// TwinCAT 3 PLC project Untitled1
// ProgramVersion: 3.1.4024.0
// libraries:
//   Tc2_MC2, * (Beckhoff Automation GmbH)
//   Tc2_Standard, * (Beckhoff Automation GmbH)
//   Tc2_System, * (Beckhoff Automation GmbH)
//   Tc3_Module, * (Beckhoff Automation GmbH)
// project tree:
//   DUTs/ ST_AchsAuftrg.TcDUT, ST_AchsFreigb.TcDUT (not stored), ST_AchsGrdfkt.TcDUT (not stored), ST_AchsInOut.TcDUT, ST_AchsKoppln.TcDUT (not stored), ST_AchsParam.TcDUT, ST_AchsStatus.TcDUT, ST_MeldServoSchrauber_1.TcDUT, ST_NcAchsen.TcDUT, ST_ParamSKSServoschrauber.TcDUT
//   GVLs/ GlobalVar_NcAchsen.TcGVL
//   / PlcTask.TcTTO (not stored)
//   POUs/10_Funktionen/Diverse/ FB_LogFile_Schrauber.TcPOU (not stored), FB_Mittelwert.TcPOU (not stored)
//   POUs/10_Funktionen/History/ FB_StepHistory.TcPOU
//   POUs/10_Funktionen/SchraubBearb/Obj/ FB_Obj_Error_Schrauber.TcPOU (not stored), FB_Obj_IOSchlauch.TcPOU (not stored)
//   POUs/ FB_Schrauber_PnP.TcPOU (not stored), FB_Schrauber_PnP_Neu.TcPOU (not stored)

// ---- DUTs/ST_AchsAuftrg.TcDUT
TYPE ST_AchsAuftrg :
STRUCT
	// Achs-Fahrauftrag
	sPTP_AuftrgTyp		:STRING(15);	// Beschreibung des Achstyp. Standard, Endlos oder Modulo
	
	bPTP_PosiFrg		:BOOL;	// Achse hat die Freigabe zu Positionieren. Betriebsbereit, beide Vorschubfreigaben und kein anderer Achsstart steht an.

	fPTP_ZielPos		:LREAL;	// aktuelle Zielposition für den Achsfahrauftrag
	fPTP_LetzZiel		:LREAL;	// Zu letzt angefahrene Zielposition
	fPTP_Geschw			:LREAL;	// in %
	ePTP_BuffMode		:MC_BufferMode;	(*MC_Aborting,
												  MC_Buffered,
												  MC_BlendingLow,
												  MC_BlendingPrevious,
												  MC_BlendingNext,
												  MC_BlendingHigh*)
	arrPTP_start		:ARRAY[1..3] OF BOOL;	// Achsstart für 3 verschiedene Betriebsmodi. Definiert in E_AchsFahrauftraege oder in NcParameter als Konstante
	bPTP_aktiv			:BOOL;	// Achsauftrag ist gestartet und auch aktiv
	bPTP_inZiel			:BOOL;	// Achsauftrag ist gestartet und im Ziel. Gibt es bei Endlosbetrieb nicht. Wird bei Verwendung vom FB_AchsStartAusf sofort wieder FALSE
	bPTP_inFenst		:BOOL;	// Achsauftrag ist gestartet und im Ziel +- 0.1 Grad oder mm. Gibt es bei Endlosbetrieb nicht.
	bPTP_stop			:BOOL;	// Achsauftrag wird gestoppt. Wird bei Verwendung vom FB_AchsStartAusf ggf. überschrieben
	bPTP_Autostop		:BOOL;	// wird aktuell nicht verwendet
	bPTP_gest			:BOOL;	// Achsauftrag wurde gestoppt. Ist nur bei aktivem bPTP_stop TRUE. Bedeutet, dass auch hier der FB_AchsStartAusf das überschreiben könnte
	bPTP_halt			:BOOL;	// Override auf 0%. Es wird mit der Beschleunigung aus dem Systemmanager gerampt
	bPTP_verz			:BOOL;	// Override auf den Wert aus der Freig-Struktur setzen.
END_STRUCT
END_TYPE

// ---- DUTs/ST_AchsInOut.TcDUT
TYPE ST_AchsInOut :
STRUCT
	
	// Eingänge
	// #######################################################################
	I_nEinspeiseStatusword			AT %I*: WORD;	(*S-0-01720.0.2
										Bit 0 - 3 	-> reserviert
										Bit 4			-> Netzspannung OK
										Bit 5			-> Hardware bereit zum Einschalten
										Bit 6			-> Zwischenkreis wird gerade geladen, oder ist geladen
										Bit 8-9		-> Rückmeldung Betriebsart
										Bit 10		-> Zwischenkreisentladung angewählt und Zwischenkreis spannungsfrei (< ca. 35 V)
										Bit 11		-> Bremswiderstand aktiv
										Bit 12		-> Warnung aktiv
										Bit 13		-> Fehler aktiv
										Bit 14		-> Bereit zur Freigabe: Netzschütz geschlossen, Zwischenkreis geladen. Die versorgten Achsen zeigen "bb".
										Bit 15		-> Die Freigabe ist gegeben, d.h. der Zwischenkreis ist belastbar. Die versorgten Achsen können nach "Ab" geschaltet werden und die Antriebsfreigabe kann gesetzt werden.
															Bei den Wechselrichtern XM* muss das Bit von der Steuerung beschrieben werden, wenn der Versorger bzw. der versorgenden Umrichter den Status "Freigabe" gesetzt hat.
										*)

	I_nDCStatusword					AT %I*: WORD;	(*P-0-0115
										Bit 0 	 	-> Antrieb Betriebsbereit
										Bit 1			-> Antrieb bereit zur Leistungsabgabe
										Bit 2			-> Warnung (ZKL 2) steht an
										Bit 3			-> Antrieb folgt (ext.) Sollwertvorgabe
										Bit 4			-> Antrieb-Halt ist aktiv und Achse ist im Stillstand
										Bit 5			-> Kommandozustand hat sich geändert
										Bit 6			-> Antrieb folgt (int.) Sollwertvorgabe der SPS
										Bit 7			-> Haupt- oder Nebenbetriebsart aktiv und Initialisierung abgeschlossen, sonst 0
										Bit 8-11		-> Istbetriebsart 
										Bit 12		-> Antrieb hat Sollwertvorgabe erreicht. (Die Bildung des Bit abhängig von der aktiven BA ist weiter unten beschrieben).
										Bit 13		-> Antriebsfehler
										Bit 14/15	-> 00: Steuer- / Leistungsteil nicht betriebsbereit z.B. Antriebsfehler oder Phase 2)
															01: Steuerteil betriebsbereit (bb)
															10: Steuer- und Leistungsteil betriebsbereit (Ab)
															11: Antrieb momentenbehaftet (AF)

										*)

	I_nDigitaleEingaenge				AT %I*: DWORD;	// Hardwareeingänge von Bosch-Rexroth. Bit .3 und .4 sind die Hardwareendlagen 
	I_nStatusHaltebremse				AT %I*: WORD;	
	I_nStatusGehaltNennmoment		AT %I*: WORD;
	I_nBetriebsstundenzaehler		AT %I*: UDINT;
	I_nDiagnoseNummer					AT %I*: DWORD;
	
	I_nDrehmomentIstwert				AT %I*: INT;	// In 0,1%. Also 1000 ist 100%
	
	I_nSignalstatuswort				AT %I*: WORD;
	
	I_nZustandsklasse3				AT %I*: WORD;
	
	// Ausgänge
	// #######################################################################
	Q_nDrehmomentGrenzwert 			AT %Q*: INT;	// Drehmoment Grenzwert Bipolar in 0,1%. Also 1000 ist 100%

	Q_nEinspeiseSteuerwort			AT %Q*: WORD;	(*S-0-01720.0.1
										Bit 0 - 7 	-> reserviert
										Bit 8-9		-> Betriebsartvorwahl
										Bit 10		-> Funktion Zwischenkreisentladung starten
										Bit 11		-> n.v.
										Bit 12		-> Betätigung des versorgerintegrierten Betriebsbereitrelais, mit dem ein optionales Hauptschütz (vorgelagertes, zusätzliches Schaltelement) freigegeben werden kann.
										Bit 13		-> Fehler aktiv
										Bit 14		-> Zwischenkreis laden und Netzschütz einschalteten - Gerät geht in Gleichrichterbetrieb
										Bit 15		-> Freigabe, Sollbetriebsart aktivieren -> Wirkt auf die IGBT-Brücke des Versorgungsgeräts, aktiviert die DC-Zwischenkreisspannungsregelung und die Sollbetriebsart
										*)

	Q_nDCPowerControl					AT %Q*: WORD;	(*S-0-0240
										Bit 0 		->Der Zwischenkreis ist bereit zur Leistungsabgabe und -aufnahme (Achse meldet antriebsbereit "Ab")
										*)

	Q_nSignalsteuerwort				AT %Q*: WORD;	(*
										Bit 0 - ReglerReset,
										Bit 1 - Fahren auf Festanschlag
										Bit 2 - Bremsentest ausführen
										*)
	
	{attribute 'TcContextName':='Task_AchsFastStop'}
	Q_bAchsNcAchsFastStop			AT %Q*: BOOL;	// Vorschlag für eine Variable verbunden mit dem Faststop aus der NC. Diese Variable hat den TcContextName: 'Task_AchsFastStop'. Dafür muss diese Task mit diesem Namen natürlich existieren.

END_STRUCT
END_TYPE

// ---- DUTs/ST_AchsParam.TcDUT
TYPE ST_AchsParam :
STRUCT
	// Achs-Parameter

	bLesSchrFrg		:BOOL;	// bei steigender Flanke werden alle Parameter gelesen und geschrieben

	bOhnSoftEndl	:BOOL;	// Softwareendlagen werden bei der Zielposition nicht überwacht.

	fSoftEndlMin	:LREAL;	// RO aktuelle Softwareendlage
	fSoftEndlMax	:LREAL;	// RO aktuelle Softwareendlage
	bSoftEndlAkt	:BOOL;	// RO Softwareendlagen sind nicht aktiv
	fEilgGeschw		:LREAL;	// RO Maximale Achsgeschwindigkeit. In mm oder ° Nicht in %

	fEndlBegrMin	:LREAL;	// WO Softwareendlage min setzen
	fEndlBegrMax	:LREAL;	// WO Softwareendlage max setzen

	fPosVerrWert	:LREAL;	// Maschinen-Parameter. Wird auf die Zielposition aufaddiert. Das gleiche wie fPosOffsWert
	fPosOffsWert	:LREAL;	// Maschinen-Parameter. Wird auf die Zielposition aufaddiert. Das gleiche wie fPosVerrWert
	fGrdstlgPos		:LREAL;	// Maschinen-Parameter. Feste Zielposition bei dem Fahrauftrag arrPTP_start[cGrundPos]
	fGeschwVorg		:LREAL;	// Maschinen-Parameter. Geschwindigkeit beim Bremse einschleifen und als Zwischenspeicher zu verwenden. Bei Fahraufträgen im AchsKtrlBaustein wird immer fPTP_Geschw genommen
	fParkPos			:LREAL;	// Maschinen-Parameter. Nur ein Zwischenspeicher.
END_STRUCT
END_TYPE

// ---- DUTs/ST_AchsStatus.TcDUT
TYPE ST_AchsStatus :
STRUCT
	// Achs-Status
	bInReferz		:BOOL;	// RO Achse ist referenziert. Vorallem bei Eilschleichachsen wichtig. (direkt aus AXISREF.Status.Homed)
	bInStillst		:BOOL;	// RO Achse steht. (direkt aus AXISREF.Status.NotMoving)
	bFahrbewAkt		:BOOL;	// RO Achse wird bewegt (Encoder) oder bewegt sich selbst (Servo). (direkt aus AXISREF.Status.Moving)
	bFaehrtPos		:BOOL;	// RO Achse wird bewegt (Encoder) oder bewegt sich selbst (Servo) positiv. (direkt aus AXISREF.Status.PositiveDirection)
	bFaehrtNeg		:BOOL;	// RO Achse wird bewegt (Encoder) oder bewegt sich selbst (Servo) negativ. (direkt aus AXISREF.Status.NegativeDirection)
	bKonstFahrt		:BOOL;	// RO Achse hat eine konstante Geschwindigkeit erreicht. (direkt aus AXISREF.Status.ConstantVelocity)
	bZielPosErr		:BOOL;	// RO Achse hat ihre Zielposition erreicht. (Genauigkeit im Systemmanager angegeben) (direkt aus AXISREF.Status.InTargetPosition)
	bZielBerErr		:BOOL;	// RO Achse hat ihr Zielfenster erreicht. (Genauigkeit im Systemmanager angegeben) (direkt aus AXISREF.Status.InPositionArea)
	
	bInGrundPos		:BOOL;	// WO Achse in Grundstellung. Muss selbst beschrieben werden

	// Hardware-Status
	bAchseBTB		:BOOL;	// RO Umrichterstatus. Wird im UniAchsAnstg, UniAntrAnstgSEW oder CtrlXGrupEinschalt gesetzt.
	bFrgSchutzBer	:BOOL;	// WO Schutzbereich für diese Achse ist freigegeben. Wichtig für Ausgabe der Hardware-Fehler
END_STRUCT
END_TYPE

// ---- DUTs/ST_MeldServoSchrauber_1.TcDUT
{attribute 'pack_mode' := '1'}
TYPE ST_MeldServoSchrauber_1 :
STRUCT
{attribute 'Message.SourceID'}
	SourceID			:DINT;
	
{attribute 'Message.SourceName'}
   SourceName		:STRING;
	
	
{attribute 'Message.Text' := '%Var1: Fehler beim Nachladen in den Schrauber! Schraube fehlt!'}//-40 Schraube fehlt	
{attribute 'Message.Info' := '}
{attribute 'Message.Type' := '7'}	
{attribute 'Message.Log'  := '1'}
{attribute 'Message.Var1' := 'sName'}
	bMeldFehlNachladen			:BOOL;
{attribute 'Message.Text' := '%Var1: Langsame Geschwindigkeit wird nicht erreicht!'}	//-45	
{attribute 'Message.Info' := '}
{attribute 'Message.Type' := '7'}	
{attribute 'Message.Log'  := '1'}
{attribute 'Message.Var1' := 'sName'}
	bMeldFehlLangsameGeschwindigkeit	:BOOL;		
{attribute 'Message.Text' := '%Var1: Schraubtiefe für Solldrehzahl wird nicht erreciht!'}	//-50	
{attribute 'Message.Info' := '}
{attribute 'Message.Type' := '7'}	
{attribute 'Message.Log'  := '1'}
{attribute 'Message.Var1' := 'sName'}
	bMeldFehlTiefeSolldrehzahl	:BOOL;		
{attribute 'Message.Text' := '%Var1: Solltiefe wird nicht erreicht!'}			//-60	
{attribute 'Message.Info' := '}
{attribute 'Message.Type' := '7'}	
{attribute 'Message.Log'  := '1'}
{attribute 'Message.Var1' := 'sName'}
	bMeldFehlSollTiefe			:BOOL;		
{attribute 'Message.Text' := '%Var1: Solltiefe wurde überschritten!'}			//-61	
{attribute 'Message.Info' := '}
{attribute 'Message.Type' := '7'}	
{attribute 'Message.Log'  := '1'}
{attribute 'Message.Var1' := 'sName'}
	bMeldFehlSollTiefeUebers	:BOOL;	
{attribute 'Message.Text' := '%Var1: Solldrehmoment wird nicht erreicht!'}	 	//-65 
{attribute 'Message.Info' := '}
{attribute 'Message.Type' := '7'}	
{attribute 'Message.Log'  := '1'}
{attribute 'Message.Var1' := 'sName'}
	bMeldFehlSollDrehmom			:BOOL;	
{attribute 'Message.Text' := '%Var1: Fehler beim heben/senken der Schrauberstange!'}//-80 	
{attribute 'Message.Info' := '}
{attribute 'Message.Type' := '7'}	
{attribute 'Message.Log'  := '1'}
{attribute 'Message.Var1' := 'sName'}
	bMeldFehlSchrauberstange			:BOOL;	
{attribute 'Message.Text' := '%Var1: Fehler beim Auswerfen!'}						//-210 	
{attribute 'Message.Info' := '}
{attribute 'Message.Type' := '7'}	
{attribute 'Message.Log'  := '1'}
{attribute 'Message.Var1' := 'sName'}
	bMeldFehlAuswerfen			:BOOL;	

{attribute 'Message.Text' := '%Var1: Schrauber ist abgewählt!'}							
{attribute 'Message.Info' := '}
{attribute 'Message.Type' := '2'}	
{attribute 'Message.Log'  := '1'}
{attribute 'Message.Var1' := 'sName'}
	bMeldSchrauberAbgewaehlt	:BOOL;
	
// aktuell nicht vorhanden
//{attribute 'Message.Text' := '%Var1: Kontrolldrehmoment wird nicht eingehalten!'}		
//{attribute 'Message.Info' := '}
//{attribute 'Message.Type' := '7'}	
//{attribute 'Message.Log'  := '1'}
//{attribute 'Message.Var1' := 'sName'}
//	bMeldFehlKontrlDrehmom		:BOOL;	
//{attribute 'Message.Text' := '%Var1: Sicherheitsverriegelung Vorsteuerzylinder, X-Position nicht im Arbeitsbereich oder abgewählt!'}		
//{attribute 'Message.Info' := '}
//{attribute 'Message.Type' := '7'}	
//{attribute 'Message.Log'  := '1'}
//{attribute 'Message.Var1' := 'sName'}
//	bMeldFehlKollision			:BOOL;	
//{attribute 'Message.Text' := '%Var1: Geberwert nicht plausibel - Prüfen, ob Schrauberstange festsitzt! Bei Wechsel bitte Referenzierfahrt starten!'}		
//{attribute 'Message.Info' := '}
//{attribute 'Message.Type' := '1'}	
//{attribute 'Message.Log'  := '1'}
//{attribute 'Message.Var1' := 'sName'}
//	bMeldFehlGeberwert			:BOOL;	
	
	sName	:STRING;

	
END_STRUCT
END_TYPE

// ---- DUTs/ST_NcAchsen.TcDUT
TYPE ST_NcAchsen :
STRUCT
	nAxNr				:INT;	// RO Achsnummer im Systemmanager
	sAxName			:STRING(31);	// RO NC-Achsname aus dem Systemmanager

	bNcFehler		:BOOL;	// RO NC hat einen Fehler
	nFehlerNr		:UDINT;	// RO NC Fehlernummer
	bBetrbBer		:BOOL;	// RO NC-Achse ist Betriebsbereit. Quasi das Häckchen. (direkt aus AXISREF.Status.Operational)
	bHwFehler		:BOOL;	// RO Umrichter ist nach Freigabe des Schutzbereiches für 5s nicht Betriebsbereit.

	fPosIstwert		:LREAL;	// RO Aktuelle Position (direkt aus AXISREF.NcToPlc.ActPos)
	fVeloIstwert	:LREAL;	// RO Aktuelle Geschwindigkeit (direkt aus AXISREF.NcToPlc.ActVelo)
	fModIstwert		:LREAL;	// RO Aktueller Modulowert (direkt aus AXISREF.NcToPlc.ModuloActPos)

	fAuftrOverride	:LREAL;	// RO Aktueller Override für den Fahrauftrag

	stStatus			:ST_AchsStatus;	// Achs-Status
	stParam			:ST_AchsParam;		// Achs-Parameter
	stFreigb			:ST_AchsFreigb;	// Achs-Freigaben
	stGrdfkt			:ST_AchsGrdfkt;	// Achs-Grundfunktionen
	stKoppln			:ST_AchsKoppln;	// Achs-Koppelfunktionen
	stAuftrg			:ST_AchsAuftrg;	// Achs-Fahrauftrag
	stMeldg			:ST_AchsMeldg;		// Achs-Meldungen
	
	stEinAusG		:ST_AchsInOut;		// Achs Ein- und Ausgangsstruktur für Bosch-Rexroth-Servos

END_STRUCT
END_TYPE

// ---- DUTs/ST_ParamSKSServoschrauber.TcDUT
{attribute 'pack_mode' := '1'}
TYPE ST_ParamSKSServoschrauber :
STRUCT	
{attribute 'MaschPara.GroupName' := 'Preset.Konstant'}
{attribute 'MaschPara.Name' := 'Anwahl Schrauber Log'}
{attribute 'MaschPara.Type' := ''}
{attribute 'MaschPara.Info' := ''}
{attribute 'MaschPara.TreeViewLayer' := '-1'}   
	bLogAnwahl						:BOOL;	
{attribute 'MaschPara.GroupName' := 'Preset.Konstant'}
{attribute 'MaschPara.Name' := 'Zeitdauer Zustellhub Schrauber '}
{attribute 'MaschPara.Type' := 'ms'}
{attribute 'MaschPara.Min' := '0'}
{attribute 'MaschPara.Max' := '5000'}
{attribute 'MaschPara.Info' := ''}
{attribute 'MaschPara.TreeViewLayer' := '-1'}   
	tParam_ZeitdZustellhubSchr	:TIME;
{attribute 'MaschPara.GroupName' := 'Preset.Konstant'}
{attribute 'MaschPara.Name' := 'Zeitdauer Schrauberhub Schrauber '}
{attribute 'MaschPara.Type' := 'ms'}
{attribute 'MaschPara.Min' := '0'}
{attribute 'MaschPara.Max' := '5000'}
{attribute 'MaschPara.Info' := ''}
{attribute 'MaschPara.TreeViewLayer' := '-1'}   
	tParam_ZeitdSchraubhubSchr	:TIME;
{attribute 'MaschPara.GroupName' := 'Preset.Konstant'}
{attribute 'MaschPara.Name' := 'Zeitdauer Laufzeitfehler Auswurfhub Schrauber '}
{attribute 'MaschPara.Type' := 'ms'}
{attribute 'MaschPara.Min' := '0'}
{attribute 'MaschPara.Max' := '5000'}
{attribute 'MaschPara.Info' := ''}
{attribute 'MaschPara.TreeViewLayer' := '-1'}   
	tParam_ZeitdAuswurfSchr	:TIME;
{attribute 'MaschPara.GroupName' := 'Preset.Konstant'}
{attribute 'MaschPara.Name' := 'Zeitdauer Laufzeitfehler Schraubtakt Schrauber '}
{attribute 'MaschPara.Type' := 'ms'}
{attribute 'MaschPara.Min' := '0'}
{attribute 'MaschPara.Max' := '5000'}
{attribute 'MaschPara.Info' := ''}
{attribute 'MaschPara.TreeViewLayer' := '-1'}   
	tParam_ZeitdSchraubTakt	:TIME;



{attribute 'MaschPara.GroupName' := 'Preset.Konstant'}
{attribute 'MaschPara.Name' := 'Solltiefe der Schrauberspitze beim Schrauben'}
{attribute 'MaschPara.Type' := 'mm im Bezug auf die Schrauberspitze'}
{attribute 'MaschPara.Min' := '-10'}
{attribute 'MaschPara.Max' := '10'}
{attribute 'MaschPara.Info' := ''}
{attribute 'MaschPara.TreeViewLayer' := '-1'} 
	fParam_Sollschraubtiefe						:LREAL;
{attribute 'MaschPara.GroupName' := 'Preset.Konstant'}
{attribute 'MaschPara.Name' := 'Solltiefe der Schrauberspitze beim Schrauben (Herdumbau)'}
{attribute 'MaschPara.Type' := 'mm im Bezug auf die Schrauberspitze'}
{attribute 'MaschPara.Min' := '0'}
{attribute 'MaschPara.Max' := '15'}
{attribute 'MaschPara.Info' := ''}
{attribute 'MaschPara.TreeViewLayer' := '-1'} 
	fParam_SollschraubtiefeHerdumbau						:LREAL;	
{attribute 'MaschPara.GroupName' := 'Preset.Konstant'}
{attribute 'MaschPara.Name' := 'Umschalttiefe ab der der Schrauber langsam dreht'}
{attribute 'MaschPara.Type' := 'mm im Bezug auf die Schrauberspitze''}
{attribute 'MaschPara.Min' := '-10'}
{attribute 'MaschPara.Max' := '100'}
{attribute 'MaschPara.Info' := ''}
{attribute 'MaschPara.TreeViewLayer' := '-1'} 
	fParam_Umschalttiefe						:LREAL;
{attribute 'MaschPara.GroupName' := 'Preset.Konstant'}
{attribute 'MaschPara.Name' := 'Tiefe ab der der Schrauber auf Solldrehzahl umschaltet'}
{attribute 'MaschPara.Type' := 'mm im Bezug auf die Schrauberspitze''}
{attribute 'MaschPara.Min' := '-10'}
{attribute 'MaschPara.Max' := '100'}
{attribute 'MaschPara.Info' := ''}
{attribute 'MaschPara.TreeViewLayer' := '-1'} 
   fSchraubTiefeSollDrehzahl			 	:LREAL;
	
{attribute 'MaschPara.GroupName' := 'Preset.Konstant'}
{attribute 'MaschPara.Name' := 'Sollmoment des Antriebes beim Schrauben'}
{attribute 'MaschPara.Type' := 'Nm'}
{attribute 'MaschPara.Min' := '-10'}
{attribute 'MaschPara.Max' := '100'}
{attribute 'MaschPara.Info' := ''}
{attribute 'MaschPara.TreeViewLayer' := '-1'} 
	fParam_Sollmoment			:LREAL;
{attribute 'MaschPara.GroupName' := 'Preset.Konstant'}
{attribute 'MaschPara.Name' := 'Solldrehzahl des Antriebes beim Schrauben'}
{attribute 'MaschPara.Type' := '% des max. Antriebsdrehzahl'}
{attribute 'MaschPara.Min' := '-10'}
{attribute 'MaschPara.Max' := '100'}
{attribute 'MaschPara.Info' := ''}
{attribute 'MaschPara.TreeViewLayer' := '-1'} 
	fParam_Solldrehzahl	:LREAL;	
{attribute 'MaschPara.GroupName' := 'Preset.Konstant'}
{attribute 'MaschPara.Name' := 'Drehzahl beim Start des Schraubvorgangs'}
{attribute 'MaschPara.Type' := '% des max. Antriebsdrehzahl'}
{attribute 'MaschPara.Min' := '-10'}
{attribute 'MaschPara.Max' := '100'}
{attribute 'MaschPara.Info' := ''}
{attribute 'MaschPara.TreeViewLayer' := '-1'} 
	fStartDrehzahl	:LREAL;	

END_STRUCT
END_TYPE

// ---- GVLs/GlobalVar_NcAchsen.TcGVL
{attribute 'Tc2GvlVarNames'}
VAR_GLOBAL
	arrNcAchsen								: ARRAY[0..2] OF ST_NcAchsen;
END_VAR

// ---- POUs/10_Funktionen/History/FB_StepHistory.TcPOU
FUNCTION_BLOCK FB_StepHistory
VAR CONSTANT
	cMaxStepHistory	:INT	:=	50;
END_VAR
VAR_INPUT
	I_nStep				:INT;
END_VAR
VAR
	n						:INT;
	arrStepHistory		:ARRAY[1..cMaxStepHistory] OF STRING(21);
	nOldHistoryStep	:INT;
END_VAR

	(***********************************************************************)
	IF	I_nStep <> nOldHistoryStep
	THEN
		FOR n := cMaxStepHistory-1  TO 1 BY -1
		DO
			arrStepHistory[n+1] 	:=	arrStepHistory[n];
		END_FOR

		arrStepHistory[1]		:=	INT_TO_STRING(I_nStep);
		FOR n := 5-LEN(arrStepHistory[1]) TO 1 BY -1
		DO
			arrStepHistory[1] := CONCAT(' ', arrStepHistory[1]);
		END_FOR
		arrStepHistory[1] := CONCAT(arrStepHistory[1], ' - ');
		arrStepHistory[1] := CONCAT(arrStepHistory[1], RIGHT(prgMAIN.fbZeitstempel.Q_objTimestamp.sQ, 12));

	END_IF

	nOldHistoryStep := I_nStep;

END_FUNCTION_BLOCK
